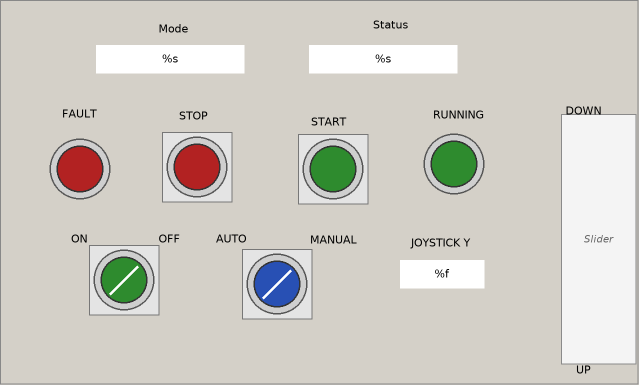
VISUALIZATION VirtualControlBox  // 639x385
    Lamp1 (419,129 70x70), variable: G_VirtualControlBox.bGreenLight, style: Lamp-Lamp1-Green
    Lamp1 (45,134 70x70), variable: G_VirtualControlBox.bRedLight, style: Lamp-Lamp1-Red
    PushSwitch (162,132 70x70), variable: G_VirtualControlBox.bStopButton, behaviour: TAP, style: Switch-PushSwitch-Red
    PushSwitch (298,134 70x70), variable: G_VirtualControlBox.bStartButton, behaviour: TAP, style: Switch-PushSwitch-Green
    RotarySwitch (89,245 70x70), variable: G_VirtualControlBox.bOnSelector, behaviour: TOGGLE, style: Switch-RotarySwitch-Green
    Label (51,224 57x30), "ON"
    Label (141,224 57x30), "OFF"
    RotarySwitch (242,249 70x70), variable: G_VirtualControlBox.bAutoSelector, behaviour: TOGGLE, style: Switch-RotarySwitch-Blue
    Label (203,224 57x30), "AUTO"
    Label (305,225 57x30), "MANUAL"
    Slider (561,114 75x250), variable: G_VirtualControlBox.fJoystickY, scale -1..1
    Label (51,99 57x30), "FAULT"
    Label (430,100 57x30), "RUNNING"
    Label (300,107 57x30), "START"
    Label (165,101 57x30), "STOP"
    Label (385,228 111x30), "JOYSTICK Y"
    Textfield (399,259 86x30), "%f", text variable: G_VirtualControlBox.fJoystickY
        OnMouseClick: write the text variable via Default, min -1, max 1
    Label (118,14 111x30), "Mode"
    Label (335,10 111x30), "Status"
    Textfield (95,44 150x30), "%s", text variable: G_Work.eMode
    Textfield (308,44 150x30), "%s", text variable: G_Work.eStatus
    Label (528,96 111x30), "DOWN"
    Label (528,355 111x30), "UP"
END_VISUALIZATION

(* stored: Version 1.1.0.1, ProductVersion 3.1.4024.10
   Visu VirtualControlBox: Id {f8cd26e7-94c0-46eb-a6ac-c63bc8ba24e3} *)
